(* PLC project Unnamed, Unknown Unnamed 1 *)
(* stored: creationDateTime 2026-04-29T12:18:43, modificationDateTime 2026-04-29T12:18:43 *)

PROGRAM main
  VAR
    LedBuiltIn AT %QX0.0 : BOOL;
  END_VAR
  VAR
    TimerOn : BOOL;
    TON0 : TON;
  END_VAR

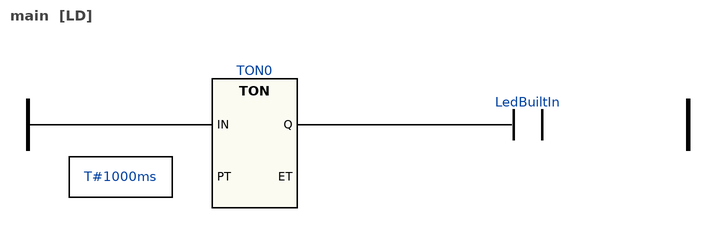
(* LD diagram, written out as Structured Text *)
TON0(IN := TRUE, PT := T#1000ms);
(* drawn but not wired to any output: LedBuiltIn *)
END_PROGRAM

CONFIGURATION Config0
  RESOURCE Res0 ON PLC
    TASK task0(INTERVAL := T#20ms, PRIORITY := 1);
    PROGRAM instance0 WITH task0 : main;
  END_RESOURCE
END_CONFIGURATION
